// Gets the lower bound index of the array of specified type.
FUNCTION F_GetLRealArrayLowerBound : T_Position // The lower bound index of the specified array.
VAR_IN_OUT
	arArray : ARRAY[*] OF LREAL; // The array to query.
END_VAR

F_GetLRealArrayLowerBound := LOWER_BOUND(arArray, 1);

END_FUNCTION

(* stored: Version 1.1.0.1
   POU F_GetLRealArrayLowerBound: Id {065dc629-dd07-0e64-2fa7-676306f8f5fc}, SpecialFunc None *)
